PROGRAM MAIN
VAR
END_VAR

P_Example_1_TONS();

END_PROGRAM

(* stored: Version 1.1.0.1, ProductVersion 3.1.4024.4
   POU MAIN: Id {d9add0bd-ac01-4108-be46-17a639b29ddc}, SpecialFunc None *)
